{attribute 'qualified_only'}
VAR_GLOBAL
	
//Atrium
	strEnOceanSwitch_AtriumNiveau_PladeB				: Tc2_EnOcean.STR_EnOceanSwitch;
	strEnOceanSwitch_AtriumNiveau_Service				: Tc2_EnOcean.STR_EnOceanSwitch;


//Gange
	strEnOceanSwitch_Rum_4_531                        : Tc2_EnOcean.STR_EnOceanSwitch;

//Rum
     strEnOceanSwitch_Rum_4_513_Indgang1_1              : Tc2_EnOcean.STR_EnOceanSwitch;
     strEnOceanSwitch_Rum_4_513_Indgang1_2              : Tc2_EnOcean.STR_EnOceanSwitch;
     strEnOceanSwitch_Rum_4_513_Indgang2                : Tc2_EnOcean.STR_EnOceanSwitch;
     strEnOceanSwitch_Rum_4_517                         : Tc2_EnOcean.STR_EnOceanSwitch;
     strEnOceanSwitch_Rum_4_521_Indgang1                : Tc2_EnOcean.STR_EnOceanSwitch;
     strEnOceanSwitch_Rum_4_521_Indgang2                : Tc2_EnOcean.STR_EnOceanSwitch;

END_VAR

(* stored: Version 1.1.0.1
   GVL GVL_EnOcean: Id {bec68ff9-8f1d-4ce1-b8b9-84de691aacc9} *)
